{attribute 'reflection'}
FUNCTION_BLOCK FB_Base
VAR
    {attribute 'instance-path'} 
    {attribute 'noinit'} 
    _InstanceName : STRING;
END_VAR

PROPERTY InstanceName : STRING
GET
InstanceName := _InstanceName;
END_GET
END_PROPERTY

END_FUNCTION_BLOCK

(* stored: Version 1.1.0.1
   POU FB_Base: Id {e546182a-9a61-412e-a041-ccf1a64e3676}, SpecialFunc None
   Property InstanceName: Id {391361aa-c916-4c61-9edb-2a54eb7a55c7}
   Get Get: Id {5ea0a207-a703-4bfa-bd47-aa2c1b3ca6bb} *)
